FUNCTION_BLOCK FB_System_Fullstand
VAR_INPUT
	bRefill : BOOL;
	fPosExt : LREAL;
END_VAR
VAR_OUTPUT
	iOut : UINT; // Fullstandssignal
END_VAR
VAR
	rPcntFillLevel : LREAL := 50.0; // Fullstand in Prozent
	iFillLevel : UINT;
	fPosExtAlt : LREAL;
	NotMoving : Bool;
END_VAR


// Auffüllen
IF bRefill THEN
	rPcntFillLevel := 100.0;
END_IF
// Füllstandsänderung durch Extruderbewegung
IF NOT notMoving THEN
	rPcntFillLevel := rPcntFillLevel - (fPosExt-fPosExtAlt)/360*0.5; // Füllstand - Grad/Umdrehung * 0,5% pro Umdrehung
END_IF

IF rPcntFillLevel < 0.0 THEN
	rPcntFillLevel := 0.0;
END_IF

iFillLevel := TO_UINT(rPcntFillLevel*1.7);

IF fPosExtAlt = fPosExt THEN
	NotMoving := TRUE;
ELSE
	NotMoving := FALSE;
END_IF

fPosExtAlt := fPosExt;

iOut := to_UINT(-65536/100 * rPcntFillLevel + 65536);

END_FUNCTION_BLOCK

(* stored: Version 1.1.0.1
   POU FB_System_Fullstand: Id {961d6cf8-3a96-4b5c-9d59-296a8dbef8ad}, SpecialFunc None *)
